FUNCTION_BLOCK Relay EXTENDS FB_ComponentBase IMPLEMENTS I_Relay
VAR
	output AT %Q* : BOOL;
	_Invert_Output	:BOOL;
END_VAR

(*
Other Diagnostics to add.
OPEN request time - Time to open
Close request time	- Time to Close.
UnCommanded move?
Duration contactor ON/OFF




*)

METHOD CyclicLogic
VAR_INPUT
END_VAR
IF NOT _InitComplete THEN
	_InitComplete := Initialize();
	RETURN;
END_IF


		
SUPER^.CyclicLogic();

//Set the current alarm severity for this module
//_CurrentAlarmSeverity := F_GetMaxSeverityRaised(Alarms := AlarmModuleAlarms, CurrentSeverity := _CurrentAlarmSeverity);
END_METHOD

METHOD FB_init : BOOL
VAR_INPUT
	bInitRetains : BOOL; // if TRUE, the retain variables are initialized (warm start / cold start)
	bInCopyCode : BOOL;  // if TRUE, the instance afterwards gets moved into the copy code (online change)
	Invert_Output	:BOOL;

END_VAR
_Invert_Output	:= Invert_Output;
//_Plusled_Output	:=Plusled_Output;
	IF _Invert_Output THEN
		output	:=TRUE;
	END_IF
END_METHOD

{attribute 'monitoring' := 'variable'}
PROPERTY OFF : BOOL
GET
{attribute 'monitoring':= 'variable'}
VAR
END_VAR
OFF := not ON;
END_GET
END_PROPERTY

{attribute 'monitoring':= 'variable'}
PROPERTY ON : BOOL
GET
IF _Invert_Output THEN
	ON :=NOT output;	
ELSIF NOT _Invert_Output THEN
	ON := output;	
END_IF
END_GET
END_PROPERTY

METHOD PUBLIC SwitchOff
VAR_INPUT
END_VAR
IF _Invert_Output THEN
	output	:=TRUE;
ELSE 
	output	:=FALSE;
END_IF
END_METHOD

METHOD PUBLIC SwitchOn
VAR_INPUT
END_VAR
IF _Invert_Output THEN
	output	:=FALSE;
ELSE 
	output	:=TRUE;
END_IF
END_METHOD

END_FUNCTION_BLOCK

(* stored: Version 1.1.0.1, ProductVersion 3.1.4024.15
   POU Relay: Id {ba806163-1640-4c19-8fe9-2ef896e165ee}, SpecialFunc None
   Folder I_CyclicFB: Id {c46f6721-c5cd-4e2b-afe2-8adddd5ccb9e}
   Method CyclicLogic: Id {971a716f-ce7c-4900-aa65-dd05304fc5bc}
   Method FB_init: Id {aa3a3794-ff3d-4001-9573-cd7e7471d4a6}
   Property OFF: Id {0ef33f7c-3686-45ee-8172-72397b494b46}
   Get Get: Id {f13f73bc-5843-4387-9c2c-4b0b92eeda5b}
   Property ON: Id {f77d2379-4503-4006-9e81-034cd1f8cb55}
   Get Get: Id {2e1a540e-5dd6-40e5-bc26-6103963af109}
   Method SwitchOff: Id {c1f9a978-7504-4168-be62-1b5cde7fccd2}
   Method SwitchOn: Id {8c3756b9-e47e-4fcc-81d5-a8a82bebf861} *)
